// TIA Portal V19 export
VAR_GLOBAL   // PLC tag table "RemoteSP"
   PB_Green_Lamp AT %Q8.0 : Bool;
   PB_Blue_Lamp AT %Q8.1 : Bool;
   TopLights_green_1500 AT %Q10.0 : Bool;   // TopLight green 1=on 0=off
   TopLights_red_1500 AT %Q10.1 : Bool;   // TopLight red 1=on 0=off
   TopLights_blue_1500 AT %Q10.2 : Bool;   // TopLight blue 1=on 0=off
   "ESTOP CH1" AT %I18.1 : Bool;
   Estop_LED AT %Q24.0 : Bool;
   "RFID_Gate CH1" AT %I18.0 : Bool;
   RFID_Gate_AUX AT %I22.2 : Bool;
END_VAR
